PROGRAM MAIN
VAR
	hr 							: HRESULT;
	fbCamera 					: FB_VN_SimpleCameraControl;
	eState 						: ETcVnCameraState;
	ipImageIn		    		: ITcVnImage;
	ipProcessedImage    		: ITcVnImage;
	ipImageInDisplay 			: ITcVnDisplayableImage;
	ipProcessedImageToDisplay 	: ITcVnDisplayableImage;
END_VAR

eState := fbCamera.GetState();

IF eState = TCVN_CS_ERROR THEN
	hr := fbCamera.Reset();
	
	ELSIF eState < TCVN_CS_ACQUIRING THEN
		hr := fbCamera.StartAcquisition();
		
		ELSIF eState = TCVN_CS_ACQUIRING THEN
			hr := fbCamera.GetCurrentImage(ipImageIn);
			
			IF SUCCEEDED(hr) AND ipImageIn <> 0 THEN
				hr := F_VN_Threshold(
				ipSrcImage      :=  ipImageIn,
				ipDestImage     :=  ipProcessedImage,
				fThreshold      :=  128, // half value range: (2^8)/2=128
				fMaxValue       :=  255, // max value of 8-bit image: (2^8)-1=255
				eThresholdType  :=  TCVN_TT_BINARY,
				hrPrev          :=  hr
			);
			hr := F_VN_TransformIntoDisplayableImage(ipProcessedImage, ipProcessedImageToDisplay, hr); //threshold Image
			hr := F_VN_TransformIntoDisplayableImage(ipImageIn, ipImageInDisplay, hr);        // raw image
			END_IF
END_IF

END_PROGRAM

(* stored: Version 1.1.0.1, ProductVersion 3.1.4024.12
   POU MAIN: Id {7df89916-5b7e-4f10-aae8-92fef7c4d085}, SpecialFunc None *)
